% RSLogix 500 project PROC1_TRIGGER_HOLDIN_INTERRUPT.RSS, saved by version 8.30.00.16 %
PROJECT "PROC1"    % processor: Bul.1763 MicroLogix 1100 Series B %

PROGRAM FILES
  LAD 2 "MAIN"  7 rungs

DATA FILES
  O0 OUTPUT  4 elements
  I1 INPUT  6 elements
  S2 STATUS  66 elements
  B3 BINARY  1 elements
  T4 TIMER  1 elements
  C5 COUNTER  1 elements
  R6 CONTROL  1 elements
  N7 INTEGER  1 elements
  F8 FLOAT  1 elements

LADDER 2 "MAIN"
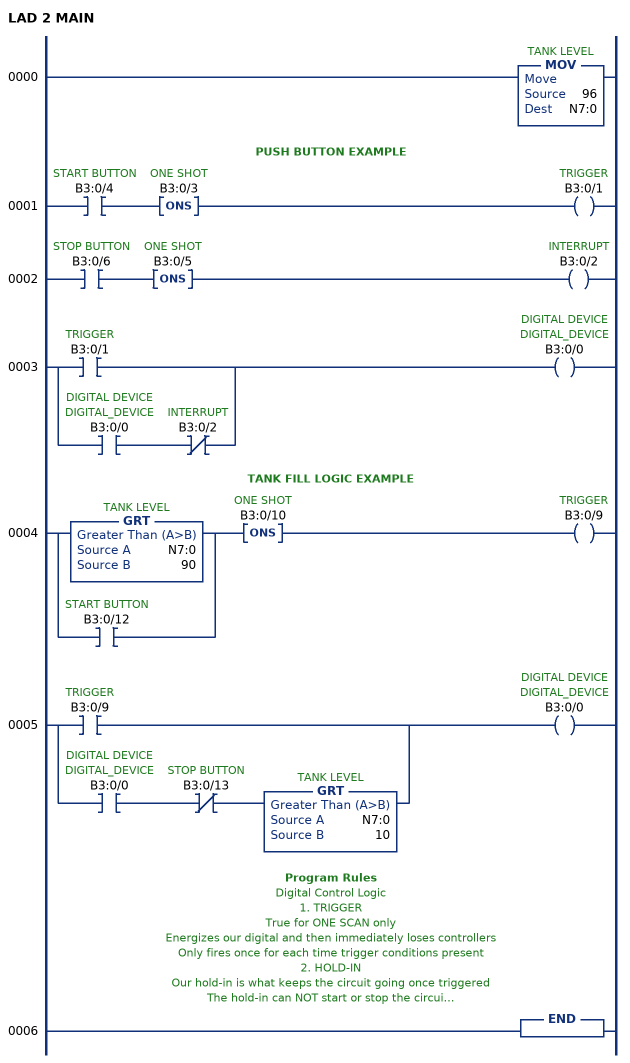
% Rung: 0 %
SOR MOV 96 N7:0 EOR
%   N7:0  "TANK LEVEL" %
% Rung: 1 %
% TITLE: PUSH BUTTON EXAMPLE %
SOR XIC B3:0/4 ONS B3:0/3 OTE B3:0/1 EOR
%   B3:0/4  "START BUTTON" %
%   B3:0/3  "ONE SHOT" %
%   B3:0/1  "TRIGGER" %
% Rung: 2 %
SOR XIC B3:0/6 ONS B3:0/5 OTE B3:0/2 EOR
%   B3:0/6  "STOP BUTTON" %
%   B3:0/5  "ONE SHOT" %
%   B3:0/2  "INTERRUPT" %
% Rung: 3 %
SOR BST XIC B3:0/1 NXB XIC B3:0/0 XIO B3:0/2 BND OTE B3:0/0 EOR
%   B3:0/1  "TRIGGER" %
%   B3:0/0  DIGITAL_DEVICE  "DIGITAL DEVICE" %
%   B3:0/2  "INTERRUPT" %
% Rung: 4 %
% TITLE: TANK FILL LOGIC EXAMPLE %
SOR BST GRT N7:0 90 NXB XIC B3:0/12 BND ONS B3:0/10 OTE B3:0/9 EOR
%   N7:0  "TANK LEVEL" %
%   B3:0/12  "START BUTTON" %
%   B3:0/10  "ONE SHOT" %
%   B3:0/9  "TRIGGER" %
% Rung: 5 %
SOR BST XIC B3:0/9 NXB XIC B3:0/0 XIO B3:0/13 GRT N7:0 10 BND OTE B3:0/0 EOR
%   B3:0/9  "TRIGGER" %
%   B3:0/0  DIGITAL_DEVICE  "DIGITAL DEVICE" %
%   B3:0/13  "STOP BUTTON" %
%   N7:0  "TANK LEVEL" %
% Rung: 6 %
% TITLE: Program Rules %
% Digital Control Logic
% 
% 1. TRIGGER
% 	True for ONE SCAN only
% 	Energizes our digital and then immediately loses controllers
% 	Only fires once for each time trigger conditions present
% 
% 2. HOLD-IN
% 	Our hold-in is what keeps the circuit going once triggered
% 	The hold-in can NOT start or stop the circuit
% 	The digital device/bit being controlled IS its own hold-in
% 
% 3. INTERRUPT
% 	A condition in series with the hold-in(same branch)
% 	Only purpose is to break continuity from the hold-in
% 	Cannot start our circuit or keep it going in any way %
SOR END EOR

REVISION NOTES
  0: Added Stop button and trigger
  1: Added Tank Level
  2: Removed GRT logic
  3: Added comments
  4: Added Tank fill logic

DATA TABLE (non-zero values as saved)
DATA N7
% N7:0 % 96
